// TIA Portal V17 export
// export: Created 2025-03-10T13:09:41.674998Z, ExportSetting WithDefaults, DisplayName Totally Integrated Automation Portal, DisplayVersion V17 Update 8, DisplayName TIA Portal Openness, DisplayVersion V17 Update 8, DisplayName TIA Portal Version Control Interface, DisplayVersion V17, DisplayName SINAMICS Startdrive Advanced, DisplayVersion V17 SP2, DisplayName SINAMICS Startdrive G110M, G120, G120C, G120D, G120P, G115D, DisplayVersion V17 SP2, DisplayName SINAMICS Startdrive G130, G150, S120, S150, SINAMICS MV, S210, DisplayVersion V17 SP2, DisplayName STEP 7 Professional, DisplayVersion V17 Update 8, DisplayName SINUMERIK ONE STEP 7 Toolbox, DisplayVersion V17 Update 12, DisplayName SINUMERIK 840D sl STEP 7 Toolbox, DisplayVersion V17 Update 12, DisplayName STEP 7 Safety, DisplayVersion V17 Update 6, DisplayName WinCC Advanced, DisplayVersion V17 Update 8
DATA_BLOCK "DB3800_UNIT_02_FIXTURE_4"   // DB3800
{ S7_Optimized_Access := 'FALSE'; DB_Accessible_From_OPC_UA := 'FALSE' }
AUTHOR : ETXETAR
VERSION : 1.0
// stored: AutoNumber false, DBAccessibleFromOPCUA false, DBAccessibleFromWebserver true, IsOnlyStoredInLoadMemory false, IsWriteProtectedInAS false
   VAR RETAIN
      INPUT_PART_A_PRESENT : Bool;   // UNIT 02 FIXTURE 4 INPUT PART A PRESENT
      INPUT_PART_B_PRESENT : Bool;   // UNIT 02 FIXTURE 4 INPUT PART B PRESENT
      INPUT_PART_C_PRESENT : Bool;   // UNIT 02 FIXTURE 4 INPUT PART C PRESENT
      INPUT_PART_D_PRESENT : Bool;   // UNIT 02 FIXTURE 4 INPUT PART D PRESENT
      INPUT_PART_A_PRESENT_FACE_N : Bool;   // UNIT 02 FIXTURE 4 INPUT PART A PRESENT FACE N UP
      INPUT_PART_B_PRESENT_FACE_N : Bool;   // UNIT 02 FIXTURE 4 INPUT PART B PRESENT FACE N UP
      INPUT_PART_C_PRESENT_FACE_N : Bool;   // UNIT 02 FIXTURE 4 INPUT PART C PRESENT FACE N UP
      INPUT_PART_D_PRESENT_FACE_N : Bool;   // UNIT 02 FIXTURE 4 INPUT PART D PRESENT FACE N UP
      INPUT_PART_A_PRESENT_FACE_R : Bool;   // UNIT 02 FIXTURE 4 INPUT PART A PRESENT FACE R UP
      INPUT_PART_B_PRESENT_FACE_R : Bool;   // UNIT 02 FIXTURE 4 INPUT PART B PRESENT FACE R UP
      INPUT_PART_C_PRESENT_FACE_R : Bool;   // UNIT 02 FIXTURE 4 INPUT PART C PRESENT FACE R UP
      INPUT_PART_D_PRESENT_FACE_R : Bool;   // UNIT 02 FIXTURE 4 INPUT PART D PRESENT FACE R UP
      INPUT_PART_A_PRESENT_MEM : Bool;   // UNIT 02 FIXTURE 4 INPUT PART A PRESENT MEMORY
      INPUT_PART_B_PRESENT_MEM : Bool;   // UNIT 02 FIXTURE 4 INPUT PART B PRESENT MEMORY
      INPUT_PART_C_PRESENT_MEM : Bool;   // UNIT 02 FIXTURE 4 INPUT PART C PRESENT MEMORY
      INPUT_PART_D_PRESENT_MEM : Bool;   // UNIT 02 FIXTURE 4 INPUT PART D PRESENT MEMORY
      INPUT_PART_A_PRESENT_FACE_N_MEM : Bool;   // UNIT 02 FIXTURE 4 INPUT PART A PRESENT FACE N UP MEMORY
      INPUT_PART_B_PRESENT_FACE_N_MEM : Bool;   // UNIT 02 FIXTURE 4 INPUT PART B PRESENT FACE N UP MEMORY
      INPUT_PART_C_PRESENT_FACE_N_MEM : Bool;   // UNIT 02 FIXTURE 4 INPUT PART C PRESENT FACE N UP MEMORY
      INPUT_PART_D_PRESENT_FACE_N_MEM : Bool;   // UNIT 02 FIXTURE 4 INPUT PART D PRESENT FACE N UP MEMORY
      INPUT_PART_A_PRESENT_FACE_R_MEM : Bool;   // UNIT 02 FIXTURE 4 INPUT PART A PRESENT FACE R UP MEMORY
      INPUT_PART_B_PRESENT_FACE_R_MEM : Bool;   // UNIT 02 FIXTURE 4 INPUT PART B PRESENT FACE R UP MEMORY
      INPUT_PART_C_PRESENT_FACE_R_MEM : Bool;   // UNIT 02 FIXTURE 4 INPUT PART C PRESENT FACE R UP MEMORY
      INPUT_PART_D_PRESENT_FACE_R_MEM : Bool;   // UNIT 02 FIXTURE 4 INPUT PART D PRESENT FACE R UP MEMORY
      CLAMPED_WITH_PART_A : Bool;   // UNIT 02 FIXTURE 4 CLAMPED WITH PART A
      CLAMPED_WITH_PART_B : Bool;   // UNIT 02 FIXTURE 4 CLAMPED WITH PART B
      CLAMPED_WITH_PART_C : Bool;   // UNIT 02 FIXTURE 4 CLAMPED WITH PART C
      CLAMPED_WITH_PART_D : Bool;   // UNIT 02 FIXTURE 4 CLAMPED WITH PART D
      CLAMPED_WITHOUT_PART_A : Bool;   // UNIT 02 FIXTURE 4 CLAMPED WITHOUT PART A
      CLAMPED_WITHOUT_PART_B : Bool;   // UNIT 02 FIXTURE 4 CLAMPED WITHOUT PART B
      CLAMPED_WITHOUT_PART_C : Bool;   // UNIT 02 FIXTURE 4 CLAMPED WITHOUT PART C
      CLAMPED_WITHOUT_PART_D : Bool;   // UNIT 02 FIXTURE 4 CLAMPED WITHOUT PART D
      CLAMPED_WITH_PARTS : Bool;   // UNIT 02 FIXTURE 4 CLAMPED WITH PARTS
      CLAMPED_WITHOUT_PARTS : Bool;   // UNIT 02 FIXTURE 4 CLAMPED WITHOUT PARTS
      PARTIAL_CLAMPED : Bool;   // UNIT 02 FIXTURE 4 PARTIAL CLAMPED
      CLAMPED_WITH_PART_ANALOG : Bool;   // UNIT 02 FIXTURE 4 CLAMPED
      CLAMPED_OK : Bool;   // UNIT 02 FIXTURE 4 CLAMPED OK
      CLAMPED_DELAYED : Bool;   // UNIT 02 FIXTURE 4 CLAMPED DELAYED
      CLAMPED_WITHOUT_PART_ANALOG : Bool;   // UNIT 02 FIXTURE 4 PARTIAL UNCLAMPED
      UNCLAMPED_ANALOG : Bool;   // UNIT 02 FIXTURE 4 UNCLAMPED
      ALL_CNC_PLC_VARIABLES_ZERO : Bool;   // UNIT 02 FIXTURE 4 ALL CNC PLC VARIABLES ZERO
      FIXTURE_NOT_CLAMPED_ALARM : Bool;   // UNIT 02 FIXTURE 4 NOT CLAMPED DURING MACHINING ALARM
      PART_A_PRESENT_DISCORDANCY : Bool;   // UNIT 02 FIXTURE 4 PART A PRESENT DISCORDANCY
      PART_B_PRESENT_DISCORDANCY : Bool;   // UNIT 02 FIXTURE 4 PART B PRESENT DISCORDANCY
      PART_C_PRESENT_DISCORDANCY : Bool;   // UNIT 02 FIXTURE 4 PART C PRESENT DISCORDANCY
      PART_D_PRESENT_DISCORDANCY : Bool;   // UNIT 02 FIXTURE 4 PART D PRESENT DISCORDANCY
      PART_A_ORIENTATED_DISCORDANCY : Bool;   // UNIT 02 FIXTURE 4 PART A ORIENTATED DISCORDANCY
      PART_B_ORIENTATED_DISCORDANCY : Bool;   // UNIT 02 FIXTURE 4 PART B ORIENTATED DISCORDANCY
      PART_C_ORIENTATED_DISCORDANCY : Bool;   // UNIT 02 FIXTURE 4 PART C ORIENTATED DISCORDANCY
      PART_D_ORIENTATED_DISCORDANCY : Bool;   // UNIT 02 FIXTURE 4 PART D ORIENTATED DISCORDANCY
      PART_TYPE_DISCORDANCY : Bool;   // UNIT 02 FIXTURE 4 PART TYPE DISCORDANCY
      ANY_PART_PRESENT : Bool;   // UNIT 02 FIXTURE 4 ANY PART PRESENT
      CLAMPED_MEMORY_DONE : Bool;   // UNIT 02 FIXTURE 4 CLAMPED MEMORY DONE
      AUX_1 : Bool;
      AUX_2 : Bool;
      AUX_3 : Bool;
      TIMER_CLAMPED_DELAY : TON_TIME;   // UNIT 02 FIXTURE 4 CLAMPED TIMER
      TIMER_PART_A_ORIENTATION { S7_SetPoint := 'True'} : TON_TIME;   // UNIT 02 FIXTURE 4 PART A ORIENTATION TIMER
      TIMER_PART_A_DISCORDANCY { S7_SetPoint := 'True'} : TON_TIME;   // UNIT 02 FIXTURE 4 PART A DISCORDANCY TIMER
      TIMER_PART_C_ORIENTATION { S7_SetPoint := 'True'} : TON_TIME;   // UNIT 02 FIXTURE 4 PART C ORIENTATION TIMER
      TIMER_PART_D_ORIENTATION { S7_SetPoint := 'True'} : TON_TIME;   // UNIT 02 FIXTURE 4 PART D ORIENTATION TIMER
      TIMER_CLAMPED_WITH_ANALOG { S7_SetPoint := 'True'} : TOF_TIME;
   END_VAR
BEGIN
   TIMER_PART_A_ORIENTATION.PT := T#200ms;
   TIMER_PART_A_DISCORDANCY.PT := T#200ms;
   TIMER_PART_C_ORIENTATION.PT := T#200ms;
   TIMER_PART_D_ORIENTATION.PT := T#200ms;
   TIMER_CLAMPED_WITH_ANALOG.PT := T#100ms;
END_DATA_BLOCK
